(* PLC project Generated.project, CODESYS CODESYS V3.5 SP19 Patch 1 *)
(* stored: creationDateTime 2026-09-14T14:47:22.327073, modificationDateTime 2026-09-14T14:47:22.327073 *)

(* ═══════════════════════════════════════════════════════════════ 🧩 ST_fbBucketCmdArbitration_Context — Contexte de gating benne ─────────────────────────────────────────────────────────────── 🎯 Rôle : Encapsuler les faits de gating consommés par FB_BucketCmdArbitration pour le séquencement couplé benne (config, intention both, état benne). Le FB dérive les flags armés (WinchBothDiveBucketOpenArmed / WinchBothAscentBucketCloseArmed) et les commandes arbitrées. 📤 Producteur : PRG_04_Treuils_Benne (câblage). 📄 Doc : DOC/AF/AF_Partie-10_Fonction_Winch_v2.1.md 🔌 État benne : 2 bits BOOL (BucketIsOpen/Closed) dérivés de _BucketState. ═══════════════════════════════════════════════════════════════ *)
TYPE ST_fbBucketCmdArbitration_Context : STRUCT
  TglEnableCoupledBucketSequencing : BOOL;  (* --> [CFG] Activation séquencement couplé benne (Commun.Cfg) *)
  MotionActive : BOOL;  (* --> [CMD] Intention mouvement both active (WinchBothMotionActive) *)
  ReqAscent : BOOL;  (* --> [CMD] Intention both montée *)
  ReqDescend : BOOL;  (* --> [CMD] Intention both descente *)
  BucketIsOpen : BOOL;  (* --> [STAT] Benne ouverte (BucketState.IsOpen) *)
  BucketIsClosed : BOOL;  (* --> [STAT] Benne fermée (BucketState.IsClosed) *)
  CoupledPhaseLocked : BOOL;  (* --> [STAT] T248 : phase couplée verrouillée (Auth.CoupledBucketPhaseLocked) -> ne PAS (ré)armer dive-open/ascent-close : plus de correction benne ni de blocage sur l'état temps réel une fois le mouvement lancé *)
END_STRUCT;
END_TYPE
